FUNCTION_BLOCK ADI_FB_CTU (* Up counter (DINT) ADI-Adapter Version *)
  (* Standard: 61499-2; Description: Copyright (c) 2026 Meisterschulen am Ostbahnhof This program and the accompanying materials are made available under the terms of the Eclipse Public License 2.0 which is available at https://www.eclipse.org/legal/epl-2.0/ SPDX-License-Identifier: EPL-2.0 NOTE: This block fires the AX output events (Q.E1, CV.E1, etc.) only on value changes using the internal E_D_FF_* change-driven wiring (e.g., E_D_FF_Q, E_D_FF_ANY_PV, E_D_FF_CU, E_D_FF_R). External filtering is no longer required. *)
  (* Version 1.0, 2026-04-21, Franz Höpfinger, Meisterschulen am Ostbahnhof, initial API and implementation and/or initial documentation *)
  PACKAGE adapter::iec61131::counters;
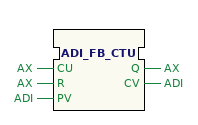
  SOCKETS
    CU : adapter::types::unidirectional::AX; (* Count up *)
    R : adapter::types::unidirectional::AX; (* Reset *)
    PV : adapter::types::unidirectional::ADI; (* Preset value *)
  END_SOCKETS
  PLUGS
    Q : adapter::types::unidirectional::AX; (* Output *)
    CV : adapter::types::unidirectional::ADI; (* Count value *)
  END_PLUGS
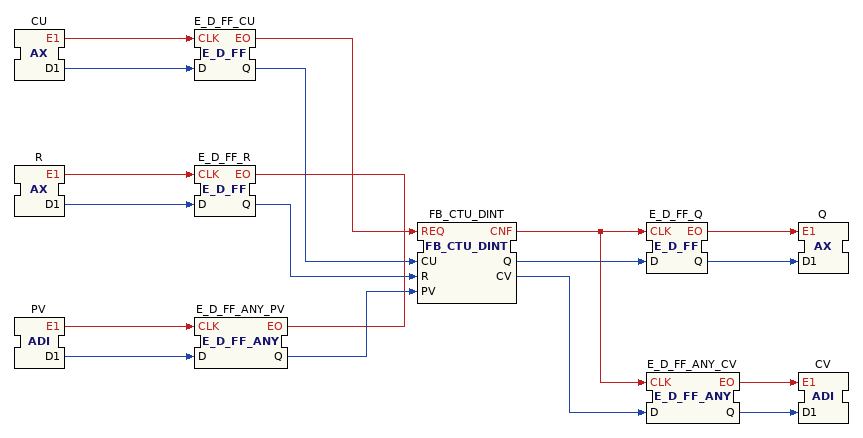
  FBS
    FB_CTU_DINT : iec61131::counters::FB_CTU_DINT;
    E_D_FF_CU : iec61499::events::E_D_FF;
    E_D_FF_R : iec61499::events::E_D_FF;
    E_D_FF_ANY_PV : iec61499::events::E_D_FF_ANY;
    E_D_FF_Q : iec61499::events::E_D_FF;
    E_D_FF_ANY_CV : iec61499::events::E_D_FF_ANY;
  END_FBS
  EVENT_CONNECTIONS
    CU.E1 TO E_D_FF_CU.CLK;
    E_D_FF_CU.EO TO FB_CTU_DINT.REQ;
    R.E1 TO E_D_FF_R.CLK;
    E_D_FF_R.EO TO FB_CTU_DINT.REQ;
    PV.E1 TO E_D_FF_ANY_PV.CLK;
    E_D_FF_ANY_PV.EO TO FB_CTU_DINT.REQ;
    FB_CTU_DINT.CNF TO E_D_FF_Q.CLK;
    E_D_FF_Q.EO TO Q.E1;
    FB_CTU_DINT.CNF TO E_D_FF_ANY_CV.CLK;
    E_D_FF_ANY_CV.EO TO CV.E1;
  END_CONNECTIONS
  DATA_CONNECTIONS
    CU.D1 TO E_D_FF_CU.D;
    E_D_FF_CU.Q TO FB_CTU_DINT.CU;
    R.D1 TO E_D_FF_R.D;
    E_D_FF_R.Q TO FB_CTU_DINT.R;
    PV.D1 TO E_D_FF_ANY_PV.D;
    E_D_FF_ANY_PV.Q TO FB_CTU_DINT.PV;
    FB_CTU_DINT.Q TO E_D_FF_Q.D;
    E_D_FF_Q.Q TO Q.D1;
    FB_CTU_DINT.CV TO E_D_FF_ANY_CV.D;
    E_D_FF_ANY_CV.Q TO CV.D1;
  END_CONNECTIONS
END_FUNCTION_BLOCK
